// TIA Portal V20 export
FUNCTION "CollectAlarms" : Void   // FC95, LAD
TITLE = Alarm Collector Unit
// Collects alarms from the respective level and categorises the alarms into the different alarm classes.
// stored: Namespace Unit1.Em4, SetENOAutomatically false
   VAR_INPUT
      resetAlarms : Bool;
      disableAlarms : Bool;
   END_VAR
   VAR_OUTPUT
      commandsToUnit : "LUC_typeStateCommands";   // Feedback to the unit
   END_VAR
   VAR CONSTANT
      DelayTime : Time := T#300ms;
      TRUE : Bool := TRUE;
      FALSE : Bool := FALSE;
   END_VAR
BEGIN

REGION Network 1: Reset Alarms
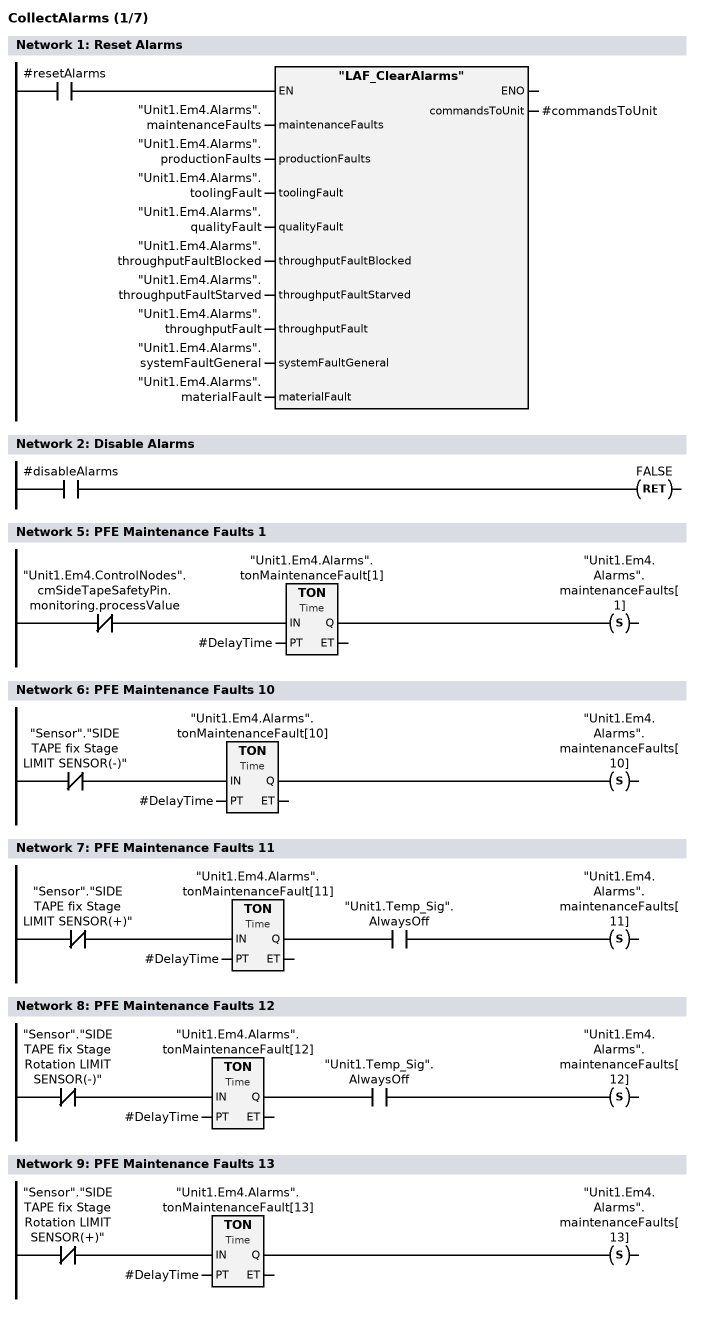
   RUNG wire#powerrail
      Contact( #resetAlarms )
      "LAF_ClearAlarms"(maintenanceFaults := "Unit1.Em4.Alarms".maintenanceFaults, productionFaults := "Unit1.Em4.Alarms".productionFaults, toolingFault := "Unit1.Em4.Alarms".toolingFault, qualityFault := "Unit1.Em4.Alarms".qualityFault, throughputFaultBlocked := "Unit1.Em4.Alarms".throughputFaultBlocked, throughputFaultStarved := "Unit1.Em4.Alarms".throughputFaultStarved, throughputFault := "Unit1.Em4.Alarms".throughputFault, systemFaultGeneral := "Unit1.Em4.Alarms".systemFaultGeneral, materialFault := "Unit1.Em4.Alarms".materialFault, commandsToUnit => #commandsToUnit)
   END_RUNG
   // the same network as SCL:
   IF #resetAlarms THEN
       "LAF_ClearAlarms"(maintenanceFaults := "Unit1.Em4.Alarms".maintenanceFaults,
                         productionFaults := "Unit1.Em4.Alarms".productionFaults,
                         toolingFault := "Unit1.Em4.Alarms".toolingFault,
                         qualityFault := "Unit1.Em4.Alarms".qualityFault,
                         throughputFaultBlocked := "Unit1.Em4.Alarms".throughputFaultBlocked,
                         throughputFaultStarved := "Unit1.Em4.Alarms".throughputFaultStarved,
                         throughputFault := "Unit1.Em4.Alarms".throughputFault,
                         systemFaultGeneral := "Unit1.Em4.Alarms".systemFaultGeneral,
                         materialFault := "Unit1.Em4.Alarms".materialFault,
                         commandsToUnit => #commandsToUnit);
   END_IF;
END_REGION

REGION Network 2: Disable Alarms
   RUNG wire#powerrail
      Contact( #disableAlarms )
      ReturnCoil( FALSE )
   END_RUNG
   // the same network as SCL:
   IF #disableAlarms THEN
       ENO := FALSE;
       RETURN;
   END_IF;
END_REGION

REGION Network 3: *************** Fault ************************
END_REGION

REGION Network 4: PFE Maintenance Faults 0
END_REGION

REGION Network 5: PFE Maintenance Faults 1
   RUNG wire#powerrail
      I_Contact( "Unit1.Em4.ControlNodes".cmSideTapeSafetyPin.monitoring.processValue )
      { S7_Templates := "time_type := Time" } "Unit1.Em4.Alarms".tonMaintenanceFault[1].TON(pt := #DelayTime, et =>)
      S_Coil( "Unit1.Em4.Alarms".maintenanceFaults[1] )
   END_RUNG
   // the same network as SCL:
   "Unit1.Em4.Alarms".tonMaintenanceFault[1].TON(IN := NOT "Unit1.Em4.ControlNodes".cmSideTapeSafetyPin.monitoring.processValue,
                           PT := #DelayTime);
   IF "Unit1.Em4.Alarms".tonMaintenanceFault[1].Q THEN
       "Unit1.Em4.Alarms".maintenanceFaults[1] := TRUE;
   END_IF;
END_REGION

REGION Network 6: PFE Maintenance Faults 10
   RUNG wire#powerrail
      I_Contact( "Sensor"."SIDE TAPE fix Stage LIMIT SENSOR(-)" )
      { S7_Templates := "time_type := Time" } "Unit1.Em4.Alarms".tonMaintenanceFault[10].TON(pt := #DelayTime, et =>)
      S_Coil( "Unit1.Em4.Alarms".maintenanceFaults[10] )
   END_RUNG
   // the same network as SCL:
   "Unit1.Em4.Alarms".tonMaintenanceFault[10].TON(IN := NOT "Sensor"."SIDE TAPE fix Stage LIMIT SENSOR(-)",
                           PT := #DelayTime);
   IF "Unit1.Em4.Alarms".tonMaintenanceFault[10].Q THEN
       "Unit1.Em4.Alarms".maintenanceFaults[10] := TRUE;
   END_IF;
END_REGION

REGION Network 7: PFE Maintenance Faults 11
   RUNG wire#powerrail
      I_Contact( "Sensor"."SIDE TAPE fix Stage LIMIT SENSOR(+)" )
      { S7_Templates := "time_type := Time" } "Unit1.Em4.Alarms".tonMaintenanceFault[11].TON(pt := #DelayTime, et =>)
      Contact( "Unit1.Temp_Sig".AlwaysOff )
      S_Coil( "Unit1.Em4.Alarms".maintenanceFaults[11] )
   END_RUNG
   // the same network as SCL:
   "Unit1.Em4.Alarms".tonMaintenanceFault[11].TON(IN := NOT "Sensor"."SIDE TAPE fix Stage LIMIT SENSOR(+)",
                           PT := #DelayTime);
   IF "Unit1.Em4.Alarms".tonMaintenanceFault[11].Q AND "Unit1.Temp_Sig".AlwaysOff THEN
       "Unit1.Em4.Alarms".maintenanceFaults[11] := TRUE;
   END_IF;
END_REGION

REGION Network 8: PFE Maintenance Faults 12
   RUNG wire#powerrail
      I_Contact( "Sensor"."SIDE TAPE fix Stage Rotation LIMIT SENSOR(-)" )
      { S7_Templates := "time_type := Time" } "Unit1.Em4.Alarms".tonMaintenanceFault[12].TON(pt := #DelayTime, et =>)
      Contact( "Unit1.Temp_Sig".AlwaysOff )
      S_Coil( "Unit1.Em4.Alarms".maintenanceFaults[12] )
   END_RUNG
   // the same network as SCL:
   "Unit1.Em4.Alarms".tonMaintenanceFault[12].TON(IN := NOT "Sensor"."SIDE TAPE fix Stage Rotation LIMIT SENSOR(-)",
                           PT := #DelayTime);
   IF "Unit1.Em4.Alarms".tonMaintenanceFault[12].Q AND "Unit1.Temp_Sig".AlwaysOff THEN
       "Unit1.Em4.Alarms".maintenanceFaults[12] := TRUE;
   END_IF;
END_REGION

REGION Network 9: PFE Maintenance Faults 13
   RUNG wire#powerrail
      I_Contact( "Sensor"."SIDE TAPE fix Stage Rotation LIMIT SENSOR(+)" )
      { S7_Templates := "time_type := Time" } "Unit1.Em4.Alarms".tonMaintenanceFault[13].TON(pt := #DelayTime, et =>)
      S_Coil( "Unit1.Em4.Alarms".maintenanceFaults[13] )
   END_RUNG
   // the same network as SCL:
   "Unit1.Em4.Alarms".tonMaintenanceFault[13].TON(IN := NOT "Sensor"."SIDE TAPE fix Stage Rotation LIMIT SENSOR(+)",
                           PT := #DelayTime);
   IF "Unit1.Em4.Alarms".tonMaintenanceFault[13].Q THEN
       "Unit1.Em4.Alarms".maintenanceFaults[13] := TRUE;
   END_IF;
END_REGION

REGION Network 10: PFE Maintenance Faults 14
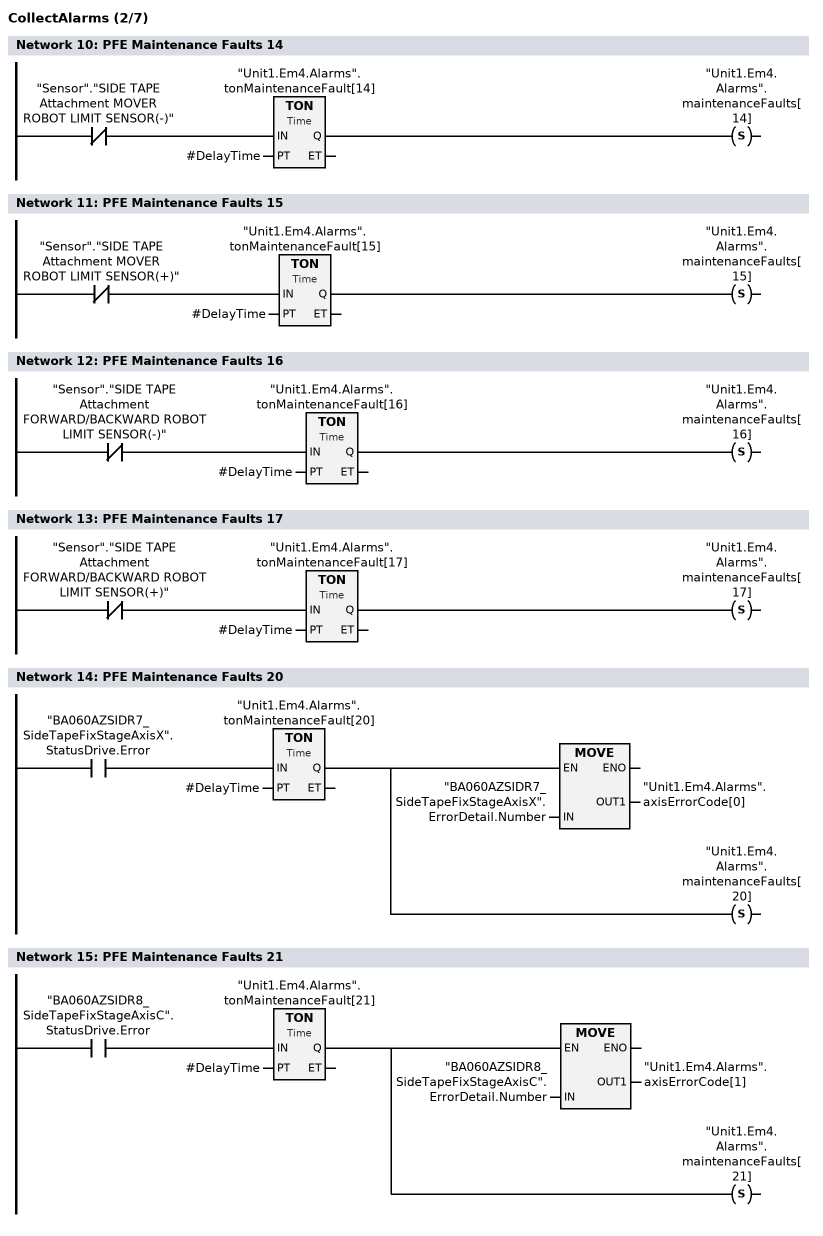
   RUNG wire#powerrail
      I_Contact( "Sensor"."SIDE TAPE Attachment MOVER ROBOT LIMIT SENSOR(-)" )
      { S7_Templates := "time_type := Time" } "Unit1.Em4.Alarms".tonMaintenanceFault[14].TON(pt := #DelayTime, et =>)
      S_Coil( "Unit1.Em4.Alarms".maintenanceFaults[14] )
   END_RUNG
   // the same network as SCL:
   "Unit1.Em4.Alarms".tonMaintenanceFault[14].TON(IN := NOT "Sensor"."SIDE TAPE Attachment MOVER ROBOT LIMIT SENSOR(-)",
                           PT := #DelayTime);
   IF "Unit1.Em4.Alarms".tonMaintenanceFault[14].Q THEN
       "Unit1.Em4.Alarms".maintenanceFaults[14] := TRUE;
   END_IF;
END_REGION

REGION Network 11: PFE Maintenance Faults 15
   RUNG wire#powerrail
      I_Contact( "Sensor"."SIDE TAPE Attachment MOVER ROBOT LIMIT SENSOR(+)" )
      { S7_Templates := "time_type := Time" } "Unit1.Em4.Alarms".tonMaintenanceFault[15].TON(pt := #DelayTime, et =>)
      S_Coil( "Unit1.Em4.Alarms".maintenanceFaults[15] )
   END_RUNG
   // the same network as SCL:
   "Unit1.Em4.Alarms".tonMaintenanceFault[15].TON(IN := NOT "Sensor"."SIDE TAPE Attachment MOVER ROBOT LIMIT SENSOR(+)",
                           PT := #DelayTime);
   IF "Unit1.Em4.Alarms".tonMaintenanceFault[15].Q THEN
       "Unit1.Em4.Alarms".maintenanceFaults[15] := TRUE;
   END_IF;
END_REGION

REGION Network 12: PFE Maintenance Faults 16
   RUNG wire#powerrail
      I_Contact( "Sensor"."SIDE TAPE Attachment FORWARD/BACKWARD ROBOT LIMIT SENSOR(-)" )
      { S7_Templates := "time_type := Time" } "Unit1.Em4.Alarms".tonMaintenanceFault[16].TON(pt := #DelayTime, et =>)
      S_Coil( "Unit1.Em4.Alarms".maintenanceFaults[16] )
   END_RUNG
   // the same network as SCL:
   "Unit1.Em4.Alarms".tonMaintenanceFault[16].TON(IN := NOT "Sensor"."SIDE TAPE Attachment FORWARD/BACKWARD ROBOT LIMIT SENSOR(-)",
                           PT := #DelayTime);
   IF "Unit1.Em4.Alarms".tonMaintenanceFault[16].Q THEN
       "Unit1.Em4.Alarms".maintenanceFaults[16] := TRUE;
   END_IF;
END_REGION

REGION Network 13: PFE Maintenance Faults 17
   RUNG wire#powerrail
      I_Contact( "Sensor"."SIDE TAPE Attachment FORWARD/BACKWARD ROBOT LIMIT SENSOR(+)" )
      { S7_Templates := "time_type := Time" } "Unit1.Em4.Alarms".tonMaintenanceFault[17].TON(pt := #DelayTime, et =>)
      S_Coil( "Unit1.Em4.Alarms".maintenanceFaults[17] )
   END_RUNG
   // the same network as SCL:
   "Unit1.Em4.Alarms".tonMaintenanceFault[17].TON(IN := NOT "Sensor"."SIDE TAPE Attachment FORWARD/BACKWARD ROBOT LIMIT SENSOR(+)",
                           PT := #DelayTime);
   IF "Unit1.Em4.Alarms".tonMaintenanceFault[17].Q THEN
       "Unit1.Em4.Alarms".maintenanceFaults[17] := TRUE;
   END_IF;
END_REGION

REGION Network 14: PFE Maintenance Faults 20
   RUNG wire#powerrail
      Contact( "BA060AZSIDR7_SideTapeFixStageAxisX".StatusDrive.Error )
      { S7_Templates := "time_type := Time" } "Unit1.Em4.Alarms".tonMaintenanceFault[20].TON(pt := #DelayTime, et =>)
      wire#w1
      Move(in := "BA060AZSIDR7_SideTapeFixStageAxisX".ErrorDetail.Number, out1 => "Unit1.Em4.Alarms".axisErrorCode[0])
   END_RUNG
   RUNG wire#w1
      S_Coil( "Unit1.Em4.Alarms".maintenanceFaults[20] )
   END_RUNG
   // the same network as SCL:
   "Unit1.Em4.Alarms".tonMaintenanceFault[20].TON(IN := "BA060AZSIDR7_SideTapeFixStageAxisX".StatusDrive.Error,
                           PT := #DelayTime);
   IF "Unit1.Em4.Alarms".tonMaintenanceFault[20].Q THEN
       "Unit1.Em4.Alarms".axisErrorCode[0] := "BA060AZSIDR7_SideTapeFixStageAxisX".ErrorDetail.Number;
       "Unit1.Em4.Alarms".maintenanceFaults[20] := TRUE;
   END_IF;
END_REGION

REGION Network 15: PFE Maintenance Faults 21
   RUNG wire#powerrail
      Contact( "BA060AZSIDR8_SideTapeFixStageAxisC".StatusDrive.Error )
      { S7_Templates := "time_type := Time" } "Unit1.Em4.Alarms".tonMaintenanceFault[21].TON(pt := #DelayTime, et =>)
      wire#w1
      Move(in := "BA060AZSIDR8_SideTapeFixStageAxisC".ErrorDetail.Number, out1 => "Unit1.Em4.Alarms".axisErrorCode[1])
   END_RUNG
   RUNG wire#w1
      S_Coil( "Unit1.Em4.Alarms".maintenanceFaults[21] )
   END_RUNG
   // the same network as SCL:
   "Unit1.Em4.Alarms".tonMaintenanceFault[21].TON(IN := "BA060AZSIDR8_SideTapeFixStageAxisC".StatusDrive.Error,
                           PT := #DelayTime);
   IF "Unit1.Em4.Alarms".tonMaintenanceFault[21].Q THEN
       "Unit1.Em4.Alarms".axisErrorCode[1] := "BA060AZSIDR8_SideTapeFixStageAxisC".ErrorDetail.Number;
       "Unit1.Em4.Alarms".maintenanceFaults[21] := TRUE;
   END_IF;
END_REGION

REGION Network 16: PFE Maintenance Faults 22
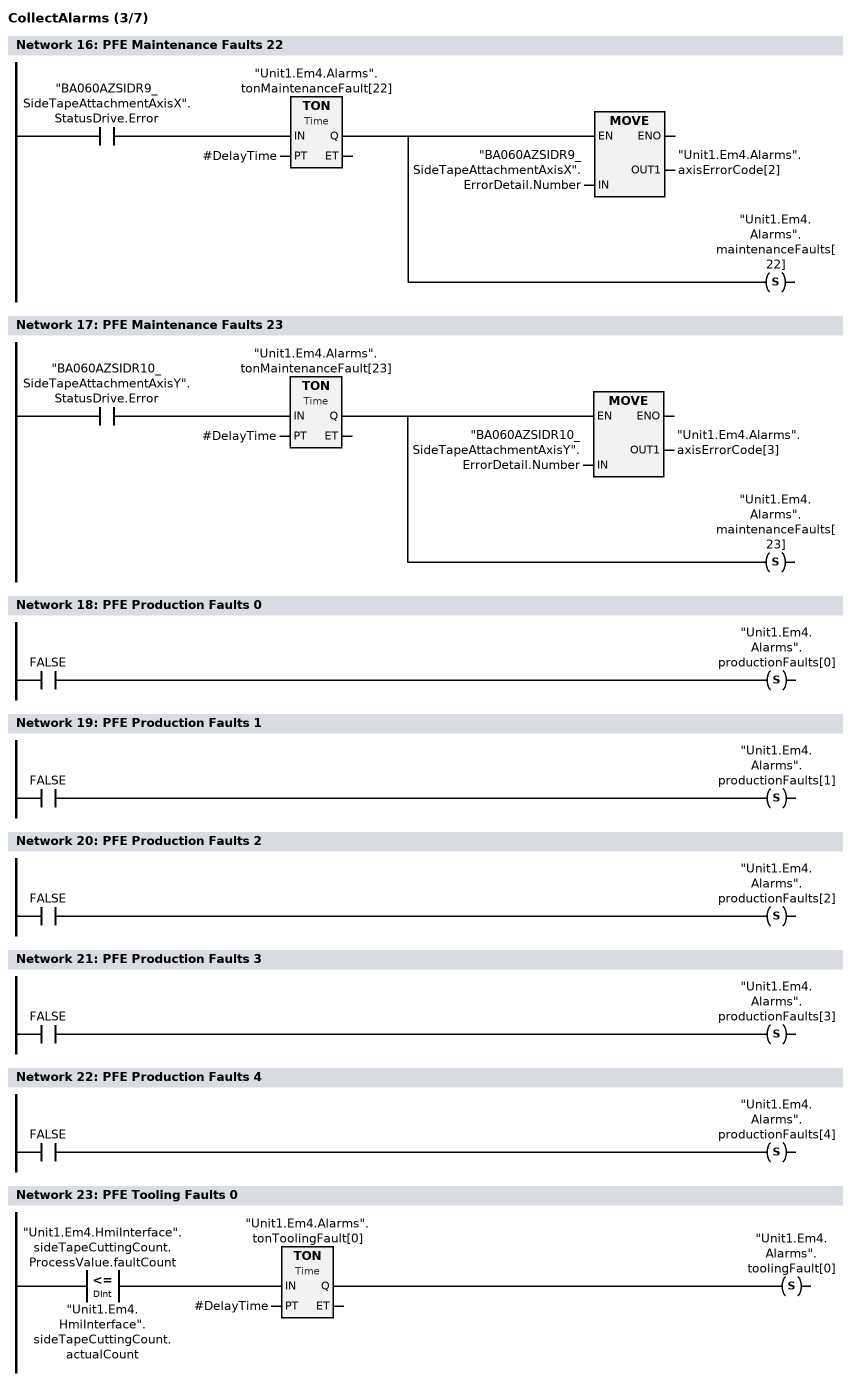
   RUNG wire#powerrail
      Contact( "BA060AZSIDR9_SideTapeAttachmentAxisX".StatusDrive.Error )
      { S7_Templates := "time_type := Time" } "Unit1.Em4.Alarms".tonMaintenanceFault[22].TON(pt := #DelayTime, et =>)
      wire#w1
      Move(in := "BA060AZSIDR9_SideTapeAttachmentAxisX".ErrorDetail.Number, out1 => "Unit1.Em4.Alarms".axisErrorCode[2])
   END_RUNG
   RUNG wire#w1
      S_Coil( "Unit1.Em4.Alarms".maintenanceFaults[22] )
   END_RUNG
   // the same network as SCL:
   "Unit1.Em4.Alarms".tonMaintenanceFault[22].TON(IN := "BA060AZSIDR9_SideTapeAttachmentAxisX".StatusDrive.Error,
                           PT := #DelayTime);
   IF "Unit1.Em4.Alarms".tonMaintenanceFault[22].Q THEN
       "Unit1.Em4.Alarms".axisErrorCode[2] := "BA060AZSIDR9_SideTapeAttachmentAxisX".ErrorDetail.Number;
       "Unit1.Em4.Alarms".maintenanceFaults[22] := TRUE;
   END_IF;
END_REGION

REGION Network 17: PFE Maintenance Faults 23
   RUNG wire#powerrail
      Contact( "BA060AZSIDR10_SideTapeAttachmentAxisY".StatusDrive.Error )
      { S7_Templates := "time_type := Time" } "Unit1.Em4.Alarms".tonMaintenanceFault[23].TON(pt := #DelayTime, et =>)
      wire#w1
      Move(in := "BA060AZSIDR10_SideTapeAttachmentAxisY".ErrorDetail.Number, out1 => "Unit1.Em4.Alarms".axisErrorCode[3])
   END_RUNG
   RUNG wire#w1
      S_Coil( "Unit1.Em4.Alarms".maintenanceFaults[23] )
   END_RUNG
   // the same network as SCL:
   "Unit1.Em4.Alarms".tonMaintenanceFault[23].TON(IN := "BA060AZSIDR10_SideTapeAttachmentAxisY".StatusDrive.Error,
                           PT := #DelayTime);
   IF "Unit1.Em4.Alarms".tonMaintenanceFault[23].Q THEN
       "Unit1.Em4.Alarms".axisErrorCode[3] := "BA060AZSIDR10_SideTapeAttachmentAxisY".ErrorDetail.Number;
       "Unit1.Em4.Alarms".maintenanceFaults[23] := TRUE;
   END_IF;
END_REGION

REGION Network 18: PFE Production Faults 0
   RUNG wire#powerrail
      Contact( FALSE )
      S_Coil( "Unit1.Em4.Alarms".productionFaults[0] )
   END_RUNG
   // the same network as SCL:
   IF FALSE THEN "Unit1.Em4.Alarms".productionFaults[0] := TRUE; END_IF;
END_REGION

REGION Network 19: PFE Production Faults 1
   RUNG wire#powerrail
      Contact( FALSE )
      S_Coil( "Unit1.Em4.Alarms".productionFaults[1] )
   END_RUNG
   // the same network as SCL:
   IF FALSE THEN "Unit1.Em4.Alarms".productionFaults[1] := TRUE; END_IF;
END_REGION

REGION Network 20: PFE Production Faults 2
   RUNG wire#powerrail
      Contact( FALSE )
      S_Coil( "Unit1.Em4.Alarms".productionFaults[2] )
   END_RUNG
   // the same network as SCL:
   IF FALSE THEN "Unit1.Em4.Alarms".productionFaults[2] := TRUE; END_IF;
END_REGION

REGION Network 21: PFE Production Faults 3
   RUNG wire#powerrail
      Contact( FALSE )
      S_Coil( "Unit1.Em4.Alarms".productionFaults[3] )
   END_RUNG
   // the same network as SCL:
   IF FALSE THEN "Unit1.Em4.Alarms".productionFaults[3] := TRUE; END_IF;
END_REGION

REGION Network 22: PFE Production Faults 4
   RUNG wire#powerrail
      Contact( FALSE )
      S_Coil( "Unit1.Em4.Alarms".productionFaults[4] )
   END_RUNG
   // the same network as SCL:
   IF FALSE THEN "Unit1.Em4.Alarms".productionFaults[4] := TRUE; END_IF;
END_REGION

REGION Network 23: PFE Tooling Faults 0
   RUNG wire#powerrail
      { S7_Templates := "SrcType := DInt" } LE_Contact(in1 := "Unit1.Em4.HmiInterface".sideTapeCuttingCount.ProcessValue.faultCount, in2 := "Unit1.Em4.HmiInterface".sideTapeCuttingCount.actualCount)
      { S7_Templates := "time_type := Time" } "Unit1.Em4.Alarms".tonToolingFault[0].TON(pt := #DelayTime, et =>)
      S_Coil( "Unit1.Em4.Alarms".toolingFault[0] )
   END_RUNG
   // the same network as SCL:
   "Unit1.Em4.Alarms".tonToolingFault[0].TON(IN := "Unit1.Em4.HmiInterface".sideTapeCuttingCount.ProcessValue.faultCount <= "Unit1.Em4.HmiInterface".sideTapeCuttingCount.actualCount,
                           PT := #DelayTime);
   IF "Unit1.Em4.Alarms".tonToolingFault[0].Q THEN "Unit1.Em4.Alarms".toolingFault[0] := TRUE; END_IF;
END_REGION

REGION Network 24: PFE Tooling Faults 1
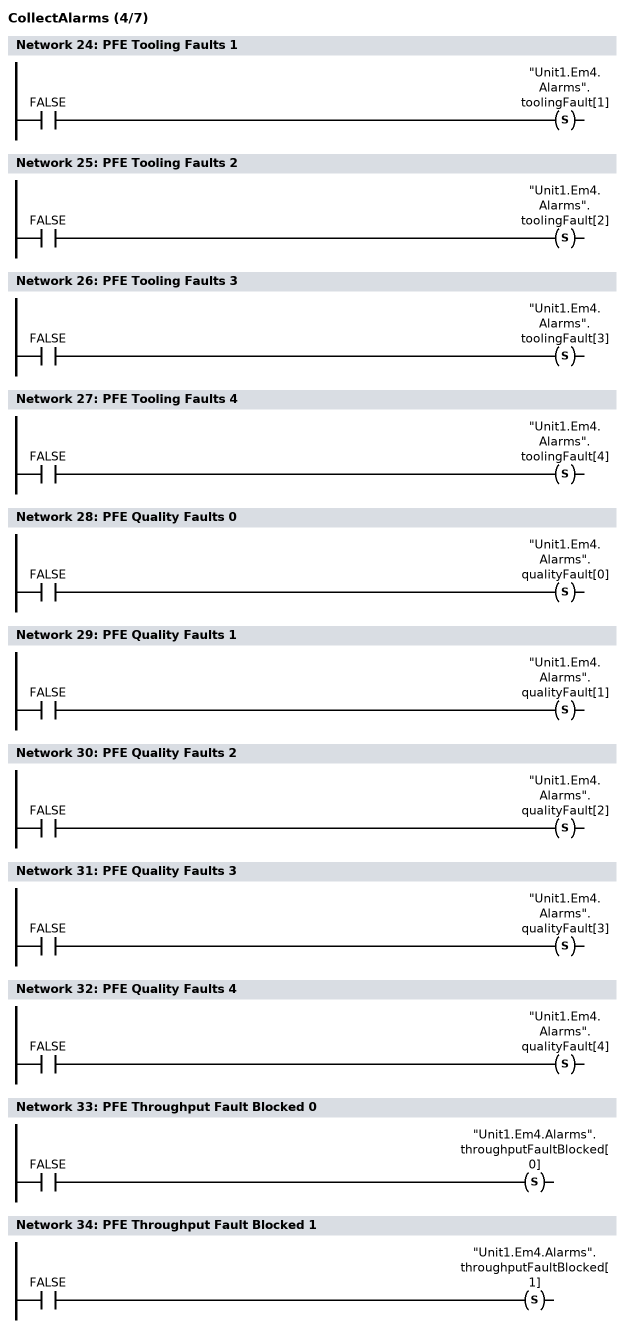
   RUNG wire#powerrail
      Contact( FALSE )
      S_Coil( "Unit1.Em4.Alarms".toolingFault[1] )
   END_RUNG
   // the same network as SCL:
   IF FALSE THEN "Unit1.Em4.Alarms".toolingFault[1] := TRUE; END_IF;
END_REGION

REGION Network 25: PFE Tooling Faults 2
   RUNG wire#powerrail
      Contact( FALSE )
      S_Coil( "Unit1.Em4.Alarms".toolingFault[2] )
   END_RUNG
   // the same network as SCL:
   IF FALSE THEN "Unit1.Em4.Alarms".toolingFault[2] := TRUE; END_IF;
END_REGION

REGION Network 26: PFE Tooling Faults 3
   RUNG wire#powerrail
      Contact( FALSE )
      S_Coil( "Unit1.Em4.Alarms".toolingFault[3] )
   END_RUNG
   // the same network as SCL:
   IF FALSE THEN "Unit1.Em4.Alarms".toolingFault[3] := TRUE; END_IF;
END_REGION

REGION Network 27: PFE Tooling Faults 4
   RUNG wire#powerrail
      Contact( FALSE )
      S_Coil( "Unit1.Em4.Alarms".toolingFault[4] )
   END_RUNG
   // the same network as SCL:
   IF FALSE THEN "Unit1.Em4.Alarms".toolingFault[4] := TRUE; END_IF;
END_REGION

REGION Network 28: PFE Quality Faults 0
   RUNG wire#powerrail
      Contact( FALSE )
      S_Coil( "Unit1.Em4.Alarms".qualityFault[0] )
   END_RUNG
   // the same network as SCL:
   IF FALSE THEN "Unit1.Em4.Alarms".qualityFault[0] := TRUE; END_IF;
END_REGION

REGION Network 29: PFE Quality Faults 1
   RUNG wire#powerrail
      Contact( FALSE )
      S_Coil( "Unit1.Em4.Alarms".qualityFault[1] )
   END_RUNG
   // the same network as SCL:
   IF FALSE THEN "Unit1.Em4.Alarms".qualityFault[1] := TRUE; END_IF;
END_REGION

REGION Network 30: PFE Quality Faults 2
   RUNG wire#powerrail
      Contact( FALSE )
      S_Coil( "Unit1.Em4.Alarms".qualityFault[2] )
   END_RUNG
   // the same network as SCL:
   IF FALSE THEN "Unit1.Em4.Alarms".qualityFault[2] := TRUE; END_IF;
END_REGION

REGION Network 31: PFE Quality Faults 3
   RUNG wire#powerrail
      Contact( FALSE )
      S_Coil( "Unit1.Em4.Alarms".qualityFault[3] )
   END_RUNG
   // the same network as SCL:
   IF FALSE THEN "Unit1.Em4.Alarms".qualityFault[3] := TRUE; END_IF;
END_REGION

REGION Network 32: PFE Quality Faults 4
   RUNG wire#powerrail
      Contact( FALSE )
      S_Coil( "Unit1.Em4.Alarms".qualityFault[4] )
   END_RUNG
   // the same network as SCL:
   IF FALSE THEN "Unit1.Em4.Alarms".qualityFault[4] := TRUE; END_IF;
END_REGION

REGION Network 33: PFE Throughput Fault Blocked 0
   RUNG wire#powerrail
      Contact( FALSE )
      S_Coil( "Unit1.Em4.Alarms".throughputFaultBlocked[0] )
   END_RUNG
   // the same network as SCL:
   IF FALSE THEN "Unit1.Em4.Alarms".throughputFaultBlocked[0] := TRUE; END_IF;
END_REGION

REGION Network 34: PFE Throughput Fault Blocked 1
   RUNG wire#powerrail
      Contact( FALSE )
      S_Coil( "Unit1.Em4.Alarms".throughputFaultBlocked[1] )
   END_RUNG
   // the same network as SCL:
   IF FALSE THEN "Unit1.Em4.Alarms".throughputFaultBlocked[1] := TRUE; END_IF;
END_REGION

REGION Network 35: PFE Throughput Fault Blocked 2
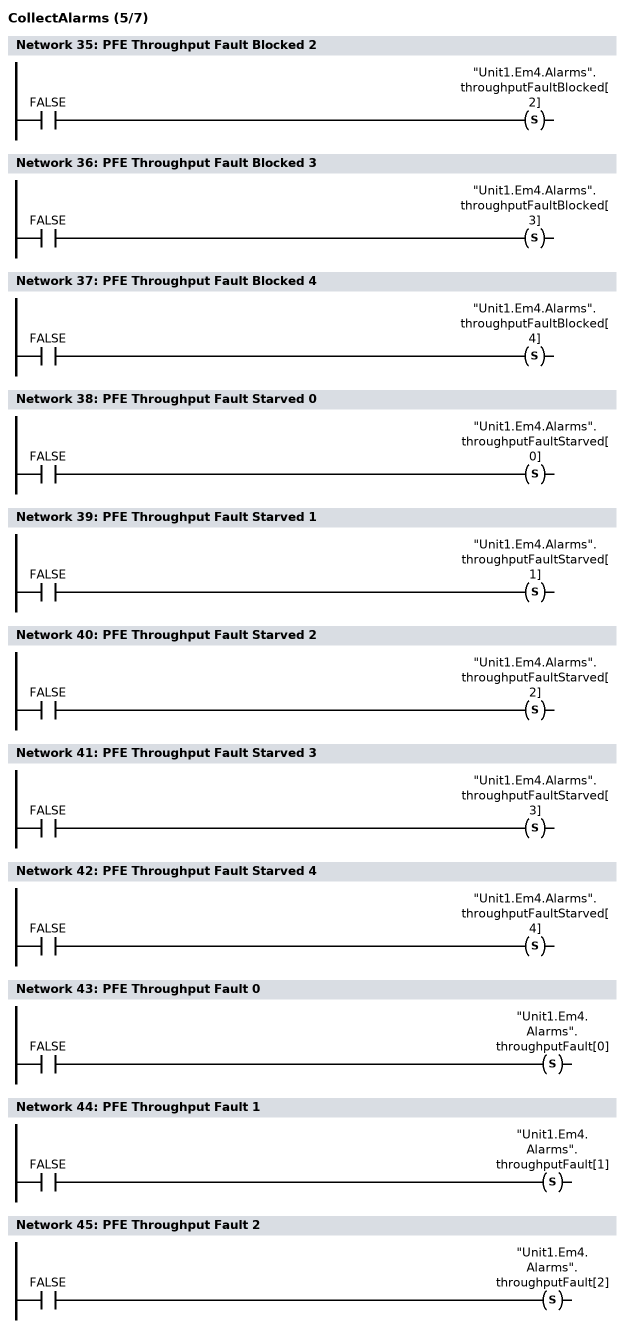
   RUNG wire#powerrail
      Contact( FALSE )
      S_Coil( "Unit1.Em4.Alarms".throughputFaultBlocked[2] )
   END_RUNG
   // the same network as SCL:
   IF FALSE THEN "Unit1.Em4.Alarms".throughputFaultBlocked[2] := TRUE; END_IF;
END_REGION

REGION Network 36: PFE Throughput Fault Blocked 3
   RUNG wire#powerrail
      Contact( FALSE )
      S_Coil( "Unit1.Em4.Alarms".throughputFaultBlocked[3] )
   END_RUNG
   // the same network as SCL:
   IF FALSE THEN "Unit1.Em4.Alarms".throughputFaultBlocked[3] := TRUE; END_IF;
END_REGION

REGION Network 37: PFE Throughput Fault Blocked 4
   RUNG wire#powerrail
      Contact( FALSE )
      S_Coil( "Unit1.Em4.Alarms".throughputFaultBlocked[4] )
   END_RUNG
   // the same network as SCL:
   IF FALSE THEN "Unit1.Em4.Alarms".throughputFaultBlocked[4] := TRUE; END_IF;
END_REGION

REGION Network 38: PFE Throughput Fault Starved 0
   RUNG wire#powerrail
      Contact( FALSE )
      S_Coil( "Unit1.Em4.Alarms".throughputFaultStarved[0] )
   END_RUNG
   // the same network as SCL:
   IF FALSE THEN "Unit1.Em4.Alarms".throughputFaultStarved[0] := TRUE; END_IF;
END_REGION

REGION Network 39: PFE Throughput Fault Starved 1
   RUNG wire#powerrail
      Contact( FALSE )
      S_Coil( "Unit1.Em4.Alarms".throughputFaultStarved[1] )
   END_RUNG
   // the same network as SCL:
   IF FALSE THEN "Unit1.Em4.Alarms".throughputFaultStarved[1] := TRUE; END_IF;
END_REGION

REGION Network 40: PFE Throughput Fault Starved 2
   RUNG wire#powerrail
      Contact( FALSE )
      S_Coil( "Unit1.Em4.Alarms".throughputFaultStarved[2] )
   END_RUNG
   // the same network as SCL:
   IF FALSE THEN "Unit1.Em4.Alarms".throughputFaultStarved[2] := TRUE; END_IF;
END_REGION

REGION Network 41: PFE Throughput Fault Starved 3
   RUNG wire#powerrail
      Contact( FALSE )
      S_Coil( "Unit1.Em4.Alarms".throughputFaultStarved[3] )
   END_RUNG
   // the same network as SCL:
   IF FALSE THEN "Unit1.Em4.Alarms".throughputFaultStarved[3] := TRUE; END_IF;
END_REGION

REGION Network 42: PFE Throughput Fault Starved 4
   RUNG wire#powerrail
      Contact( FALSE )
      S_Coil( "Unit1.Em4.Alarms".throughputFaultStarved[4] )
   END_RUNG
   // the same network as SCL:
   IF FALSE THEN "Unit1.Em4.Alarms".throughputFaultStarved[4] := TRUE; END_IF;
END_REGION

REGION Network 43: PFE Throughput Fault 0
   RUNG wire#powerrail
      Contact( FALSE )
      S_Coil( "Unit1.Em4.Alarms".throughputFault[0] )
   END_RUNG
   // the same network as SCL:
   IF FALSE THEN "Unit1.Em4.Alarms".throughputFault[0] := TRUE; END_IF;
END_REGION

REGION Network 44: PFE Throughput Fault 1
   RUNG wire#powerrail
      Contact( FALSE )
      S_Coil( "Unit1.Em4.Alarms".throughputFault[1] )
   END_RUNG
   // the same network as SCL:
   IF FALSE THEN "Unit1.Em4.Alarms".throughputFault[1] := TRUE; END_IF;
END_REGION

REGION Network 45: PFE Throughput Fault 2
   RUNG wire#powerrail
      Contact( FALSE )
      S_Coil( "Unit1.Em4.Alarms".throughputFault[2] )
   END_RUNG
   // the same network as SCL:
   IF FALSE THEN "Unit1.Em4.Alarms".throughputFault[2] := TRUE; END_IF;
END_REGION

REGION Network 46: PFE Throughput Fault 3
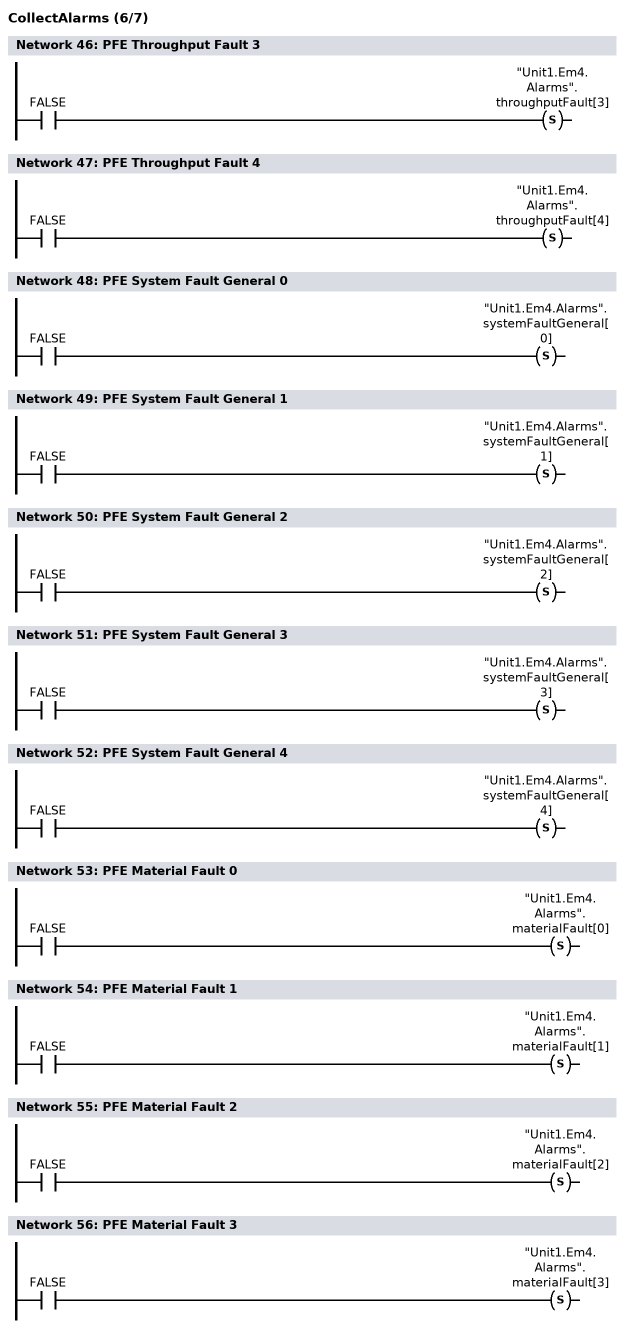
   RUNG wire#powerrail
      Contact( FALSE )
      S_Coil( "Unit1.Em4.Alarms".throughputFault[3] )
   END_RUNG
   // the same network as SCL:
   IF FALSE THEN "Unit1.Em4.Alarms".throughputFault[3] := TRUE; END_IF;
END_REGION

REGION Network 47: PFE Throughput Fault 4
   RUNG wire#powerrail
      Contact( FALSE )
      S_Coil( "Unit1.Em4.Alarms".throughputFault[4] )
   END_RUNG
   // the same network as SCL:
   IF FALSE THEN "Unit1.Em4.Alarms".throughputFault[4] := TRUE; END_IF;
END_REGION

REGION Network 48: PFE System Fault General 0
   RUNG wire#powerrail
      Contact( FALSE )
      S_Coil( "Unit1.Em4.Alarms".systemFaultGeneral[0] )
   END_RUNG
   // the same network as SCL:
   IF FALSE THEN "Unit1.Em4.Alarms".systemFaultGeneral[0] := TRUE; END_IF;
END_REGION

REGION Network 49: PFE System Fault General 1
   RUNG wire#powerrail
      Contact( FALSE )
      S_Coil( "Unit1.Em4.Alarms".systemFaultGeneral[1] )
   END_RUNG
   // the same network as SCL:
   IF FALSE THEN "Unit1.Em4.Alarms".systemFaultGeneral[1] := TRUE; END_IF;
END_REGION

REGION Network 50: PFE System Fault General 2
   RUNG wire#powerrail
      Contact( FALSE )
      S_Coil( "Unit1.Em4.Alarms".systemFaultGeneral[2] )
   END_RUNG
   // the same network as SCL:
   IF FALSE THEN "Unit1.Em4.Alarms".systemFaultGeneral[2] := TRUE; END_IF;
END_REGION

REGION Network 51: PFE System Fault General 3
   RUNG wire#powerrail
      Contact( FALSE )
      S_Coil( "Unit1.Em4.Alarms".systemFaultGeneral[3] )
   END_RUNG
   // the same network as SCL:
   IF FALSE THEN "Unit1.Em4.Alarms".systemFaultGeneral[3] := TRUE; END_IF;
END_REGION

REGION Network 52: PFE System Fault General 4
   RUNG wire#powerrail
      Contact( FALSE )
      S_Coil( "Unit1.Em4.Alarms".systemFaultGeneral[4] )
   END_RUNG
   // the same network as SCL:
   IF FALSE THEN "Unit1.Em4.Alarms".systemFaultGeneral[4] := TRUE; END_IF;
END_REGION

REGION Network 53: PFE Material Fault 0
   RUNG wire#powerrail
      Contact( FALSE )
      S_Coil( "Unit1.Em4.Alarms".materialFault[0] )
   END_RUNG
   // the same network as SCL:
   IF FALSE THEN "Unit1.Em4.Alarms".materialFault[0] := TRUE; END_IF;
END_REGION

REGION Network 54: PFE Material Fault 1
   RUNG wire#powerrail
      Contact( FALSE )
      S_Coil( "Unit1.Em4.Alarms".materialFault[1] )
   END_RUNG
   // the same network as SCL:
   IF FALSE THEN "Unit1.Em4.Alarms".materialFault[1] := TRUE; END_IF;
END_REGION

REGION Network 55: PFE Material Fault 2
   RUNG wire#powerrail
      Contact( FALSE )
      S_Coil( "Unit1.Em4.Alarms".materialFault[2] )
   END_RUNG
   // the same network as SCL:
   IF FALSE THEN "Unit1.Em4.Alarms".materialFault[2] := TRUE; END_IF;
END_REGION

REGION Network 56: PFE Material Fault 3
   RUNG wire#powerrail
      Contact( FALSE )
      S_Coil( "Unit1.Em4.Alarms".materialFault[3] )
   END_RUNG
   // the same network as SCL:
   IF FALSE THEN "Unit1.Em4.Alarms".materialFault[3] := TRUE; END_IF;
END_REGION

REGION Network 57: PFE Material Fault 4
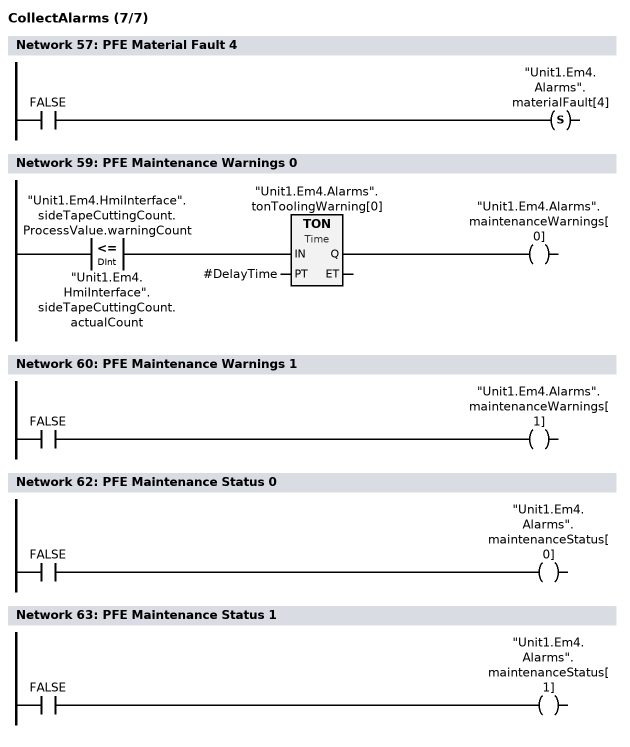
   RUNG wire#powerrail
      Contact( FALSE )
      S_Coil( "Unit1.Em4.Alarms".materialFault[4] )
   END_RUNG
   // the same network as SCL:
   IF FALSE THEN "Unit1.Em4.Alarms".materialFault[4] := TRUE; END_IF;
END_REGION

REGION Network 58: ******************** Warning ********************
END_REGION

REGION Network 59: PFE Maintenance Warnings 0
   RUNG wire#powerrail
      { S7_Templates := "SrcType := DInt" } LE_Contact(in1 := "Unit1.Em4.HmiInterface".sideTapeCuttingCount.ProcessValue.warningCount, in2 := "Unit1.Em4.HmiInterface".sideTapeCuttingCount.actualCount)
      { S7_Templates := "time_type := Time" } "Unit1.Em4.Alarms".tonToolingWarning[0].TON(pt := #DelayTime, et =>)
      Coil( "Unit1.Em4.Alarms".maintenanceWarnings[0] )
   END_RUNG
   // the same network as SCL:
   "Unit1.Em4.Alarms".tonToolingWarning[0].TON(IN := "Unit1.Em4.HmiInterface".sideTapeCuttingCount.ProcessValue.warningCount <= "Unit1.Em4.HmiInterface".sideTapeCuttingCount.actualCount,
                           PT := #DelayTime);
   "Unit1.Em4.Alarms".maintenanceWarnings[0] := "Unit1.Em4.Alarms".tonToolingWarning[0].Q;
END_REGION

REGION Network 60: PFE Maintenance Warnings 1
   RUNG wire#powerrail
      Contact( FALSE )
      Coil( "Unit1.Em4.Alarms".maintenanceWarnings[1] )
   END_RUNG
   // the same network as SCL:
   "Unit1.Em4.Alarms".maintenanceWarnings[1] := FALSE;
END_REGION

REGION Network 61: ******************** Status ********************
END_REGION

REGION Network 62: PFE Maintenance Status 0
   RUNG wire#powerrail
      Contact( FALSE )
      Coil( "Unit1.Em4.Alarms".maintenanceStatus[0] )
   END_RUNG
   // the same network as SCL:
   "Unit1.Em4.Alarms".maintenanceStatus[0] := FALSE;
END_REGION

REGION Network 63: PFE Maintenance Status 1
   RUNG wire#powerrail
      Contact( FALSE )
      Coil( "Unit1.Em4.Alarms".maintenanceStatus[1] )
   END_RUNG
   // the same network as SCL:
   "Unit1.Em4.Alarms".maintenanceStatus[1] := FALSE;
END_REGION
END_FUNCTION
